KUKA KRL program: St1_Job3_Side1.src, St1_Job3_Side1.dat

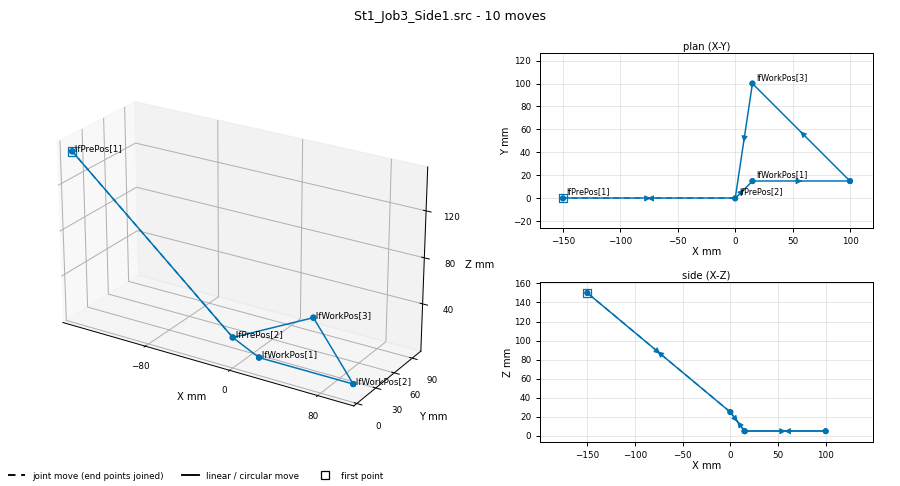
[picture p0: tool path of St1_Job3_Side1.src, 10 of 14 moves have a stored position in this frame; points joined in program order, loops and branches not executed]
--- St1_Job3_Side1.src ---
&ACCESS RVEO
&REL 3
DEF  St1_Job3_Side1 (lnActSt :IN)
   INT lnActSt,lnUsedBase,lnUsedTool
   INT lnJobNr

   ;FOLD INIT
      CONTINUE
      IF ($T1 OR $T2)THEN
         GLOBAL INTERRUPT DECL 3 WHEN $STOPMESS==TRUE DO IR_STOPM ( )
         INTERRUPT ON 3
         BAS (#INITMOV,0)
         lnActSt = 1
         PTP $POS_ACT
      ENDIF
      lnJobNr = gnJobNr3
      lnUsedBase = lnActSt + 10
      lnUsedTool = 20

      gfMillingOffset = $NULLFRAME
      gfMillingOffset.Z = -(grCuttingDepth*(gnMillingCounter-1))

      BASE_DATA[lnUsedBase] = BASE_DATA[lnActSt]:gfBaseShift[lnActSt]:gfMillingOffset
      TOOL_DATA[lnUsedTool] = TOOL_DATA[11] :{X 0,Y 0,Z 0,A 0,B 0,C 0}
   ;ENDFOLD
   REPEAT
      CONTINUE
   UNTIL (DI_SpindleStandsStill) OR NOT WatchDog(gnTimerWatchDog, 30000)

   CONTINUE
   IF NOT (DI_SpindleStandsStill) THEN
      MsgNotify("Station1/St1_Job3_Side1() -> TimeOut: Spindle speed Not StandStill")
      SpindleStop()
      gbRecoveryNeeded = TRUE
      RETURN
   ENDIF

   gbJob3StartedSt[1] = TRUE
   gbJob3DoneSt[1]    = FALSE

   MoveSettings(lnUsedBase, lnUsedTool, 100, 500)
   PTP lfPrePos[1] C_DIS
   MoveSettings(lnUsedBase, lnUsedTool, 100, 200)
   LIN lfPrePos[2] C_DIS

   ;Measure P1
   MoveSettings(lnUsedBase, lnUsedTool, 100, 200)
   LIN lfWorkPos[1]
   MoveSettings(lnUsedBase, lnUsedTool, 100, 2)
   LIN lfWorkPos[1]:{X 0.0,Y 0.0,Z -4,A 0.0,B 0.0,C 0.0}
   MoveSettings(lnUsedBase, lnUsedTool, 100, 200)
   LIN lfWorkPos[1] C_DIS
   ;Measure P2
   MoveSettings(lnUsedBase, lnUsedTool, 100, 200)
   LIN lfWorkPos[2]
   MoveSettings(lnUsedBase, lnUsedTool, 100, 2)
   LIN lfWorkPos[2]:{X 0.0,Y 0.0,Z -4,A 0.0,B 0.0,C 0.0}
   MoveSettings(lnUsedBase, lnUsedTool, 100, 200)
   LIN lfWorkPos[2] C_DIS
   ;Measure P3
   MoveSettings(lnUsedBase, lnUsedTool, 100, 200)
   LIN lfWorkPos[3]
   MoveSettings(lnUsedBase, lnUsedTool, 100, 2)
   LIN lfWorkPos[3]:{X 0.0,Y 0.0,Z -4,A 0.0,B 0.0,C 0.0}
   MoveSettings(lnUsedBase, lnUsedTool, 100, 200)
   LIN lfWorkPos[3] C_DIS
   ;END OF MEASUREMENT

   MoveSettings(lnUsedBase, lnUsedTool, 100, 200)
   TRIGGER WHEN DISTANCE=0 DELAY=0 DO endOfJob() PRIO=-1
   LIN lfPrePos[2] C_DIS
   MoveSettings(lnUsedBase, lnUsedTool, 100, 200)

   PTP lfPrePos[1] C_PTP
   MoveToPrepos(lnActSt)
END

DEF endOfJob()
   gbJob3StartedSt[1] = FALSE
   gbJob3DoneSt[1]    = TRUE
END

--- St1_Job3_Side1.dat ---
&ACCESS RVEO
&REL 3
DEFDAT  St1_Job3_Side1

   DECL FRAME lfPrePos[3]
   lfPrePos[1]={X -150.000,Y 0.0,Z 150.000,A 0.0,B 0.0,C 0.0}
   lfPrePos[2]={X 0.0,Y 0.0,Z 25.0,A 0.0,B 0.0,C 0.0}
   lfPrePos[3]={X 0.0,Y 0.0,Z 0.0,A 0.0,B 0.0,C 0.0}

   DECL FRAME lfWorkPos[12]
   lfWorkPos[1]={X 15,Y 15.0,Z 5.000,A 0.0,B 0.0,C 0.0}
   lfWorkPos[2]={X 100.0,Y 15.0,Z 5.0000,A 0.0,B 0.0,C 0.0}
   lfWorkPos[3]={X 15.0,Y 100.0,Z 5.0000,A 0.0,B 0.0,C 0.0}
   ;lfWorkPos[4]={X 100.0,Y -5.0,Z 5.0000,A 0.0,B 0.0,C 0.0}
   ;lfWorkPos[5]={X 100.0,Y 10.0,Z 5.0000,A 0.0,B 0.0,C 0.0}
   ;lfWorkPos[6]={X 10.0,Y 10.0,Z 5.0000,A 0.0,B 0.0,C 0.0}
   ;lfWorkPos[7]={X -5.0,Y 10.0,Z 5.0000,A 0.0,B 0.0,C 0.0}
   ;lfWorkPos[8]={X -5.0,Y 10.0,Z -10.000,A 0.0,B 0.0,C 0.0}
   ;lfWorkPos[9]={X -5.0,Y 100.0,Z -10.000,A 0.0,B 0.0,C 0.0}
   ;lfWorkPos[10]={X -5.0,Y 100.0,Z 5.000,A 0.0,B 0.0,C 0.0}
   ;lfWorkPos[11]={X 10.0,Y 100.0,Z 5.000,A 0.0,B 0.0,C 0.0}
   ;lfWorkPos[12]={X 10.0,Y 10.0,Z 5.000,A 0.0,B 0.0,C 0.0}


ENDDAT
